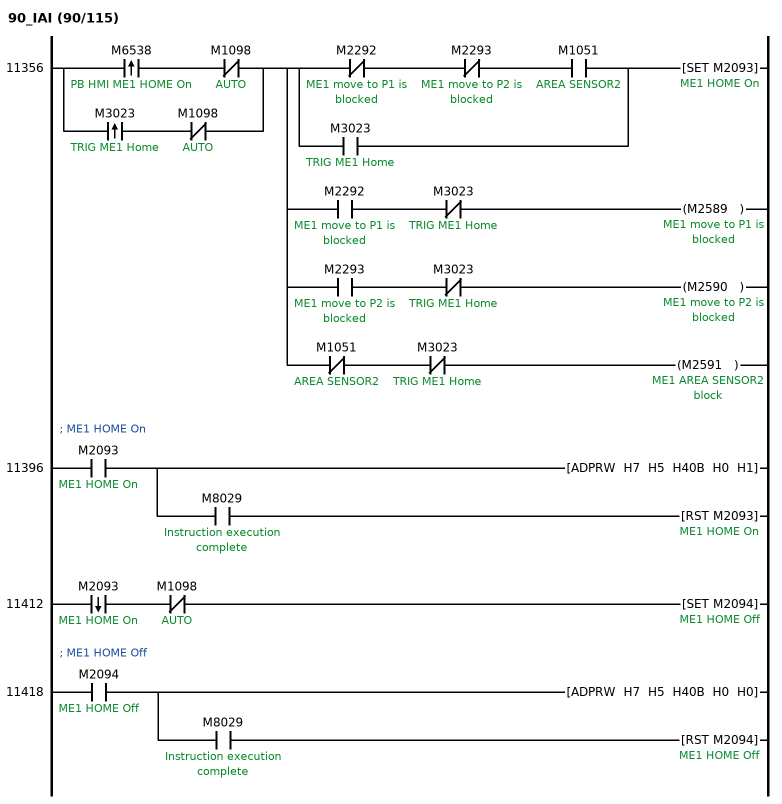
[picture p192: ladder of 90_IAI, rungs at steps 11356 to 11418]
11356 LDP     M6538  ; PB HMI ME1 HOME On
      ANI     M1098  ; AUTO
      LDP     M3023  ; TRIG ME1 Home
      ANI     M1098  ; AUTO
      ORB
      MPS
      LDI     M2292  ; ME1 move to P1 is blocked
      ANI     M2293  ; ME1 move to P2 is blocked
      AND     M1051  ; AREA SENSOR2
      OR      M3023  ; TRIG ME1 Home
      ANB
      SET     M2093  ; ME1 HOME On
      MRD
      AND     M2292  ; ME1 move to P1 is blocked
      ANI     M3023  ; TRIG ME1 Home
      OUT     M2589  ; ME1 move to P1 is blocked
      MRD
      AND     M2293  ; ME1 move to P2 is blocked
      ANI     M3023  ; TRIG ME1 Home
      OUT     M2590  ; ME1 move to P2 is blocked
      MPP
      ANI     M1051  ; AREA SENSOR2
      ANI     M3023  ; TRIG ME1 Home
      OUT     M2591  ; ME1 AREA SENSOR2 block
; ME1 HOME On
11396 LD      M2093  ; ME1 HOME On
      ADPRW   H7 H5 H40B H0 H1
      AND     M8029  ; Instruction execution complete
      RST     M2093  ; ME1 HOME On
11412 LDF     M2093  ; ME1 HOME On
      ANI     M1098  ; AUTO
      SET     M2094  ; ME1 HOME Off
; ME1 HOME Off
11418 LD      M2094  ; ME1 HOME Off
      ADPRW   H7 H5 H40B H0 H0
      AND     M8029  ; Instruction execution complete
      RST     M2094  ; ME1 HOME Off
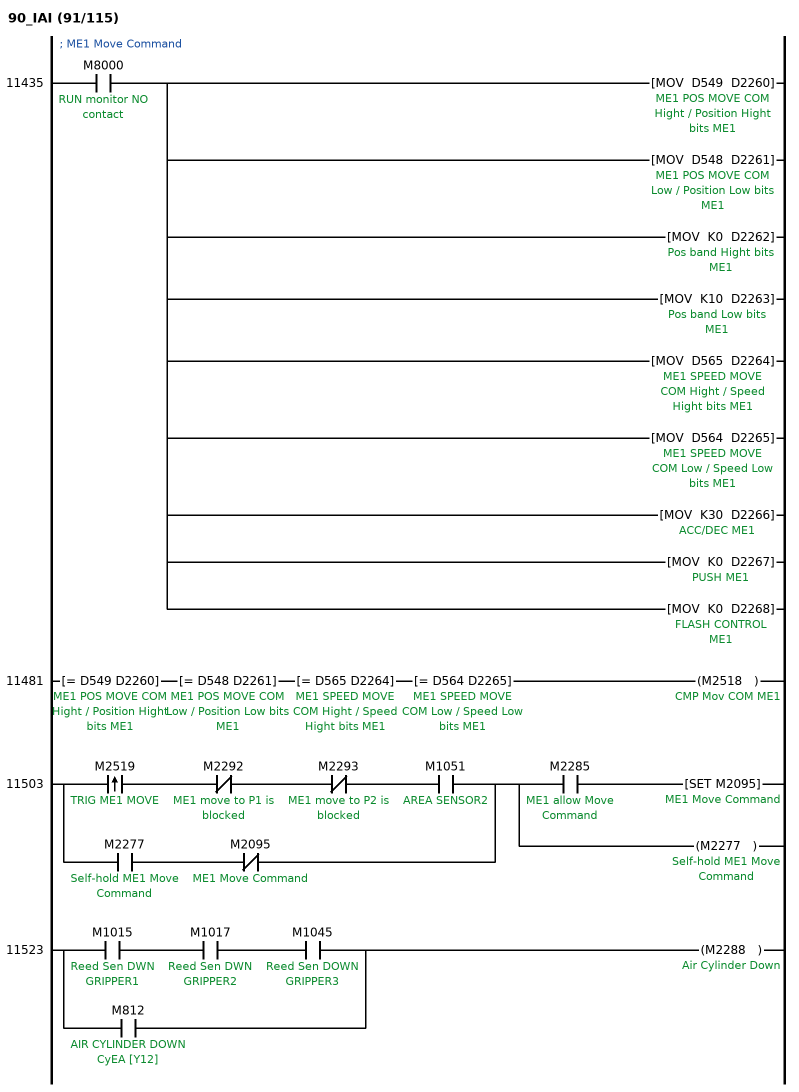
; ME1 Move Command
11435 LD      M8000  ; RUN monitor NO contact
      MOV     D549 D2260  ; ME1 POS MOVE COM Hight / Position Hight bits ME1
      MOV     D548 D2261  ; ME1 POS MOVE COM Low / Position Low bits ME1
      MOV     K0 D2262  ; Pos band Hight bits ME1
      MOV     K10 D2263  ; Pos band Low bits ME1
      MOV     D565 D2264  ; ME1 SPEED MOVE COM Hight / Speed Hight bits ME1
      MOV     D564 D2265  ; ME1 SPEED MOVE COM Low / Speed Low bits ME1
      MOV     K30 D2266  ; ACC/DEC ME1
      MOV     K0 D2267  ; PUSH ME1
      MOV     K0 D2268  ; FLASH CONTROL ME1
11481 LD=     D549 D2260  ; ME1 POS MOVE COM Hight / Position Hight bits ME1
      AND=    D548 D2261  ; ME1 POS MOVE COM Low / Position Low bits ME1
      AND=    D565 D2264  ; ME1 SPEED MOVE COM Hight / Speed Hight bits ME1
      AND=    D564 D2265  ; ME1 SPEED MOVE COM Low / Speed Low bits ME1
      OUT     M2518  ; CMP Mov COM ME1
11503 LDP     M2519  ; TRIG ME1 MOVE
      ANI     M2292  ; ME1 move to P1 is blocked
      ANI     M2293  ; ME1 move to P2 is blocked
      AND     M1051  ; AREA SENSOR2
      LD      M2277  ; Self-hold ME1 Move Command
      ANI     M2095  ; ME1 Move Command
      ORB
      MPS
      AND     M2285  ; ME1 allow Move Command
      SET     M2095  ; ME1 Move Command
      MPP
      OUT     M2277  ; Self-hold ME1 Move Command
11523 LD      M1015  ; Reed Sen DWN GRIPPER1
      AND     M1017  ; Reed Sen DWN GRIPPER2
      AND     M1045  ; Reed Sen DOWN GRIPPER3
      OR      M812  ; AIR CYLINDER DOWN CyEA [Y12]
      OUT     M2288  ; Air Cylinder Down
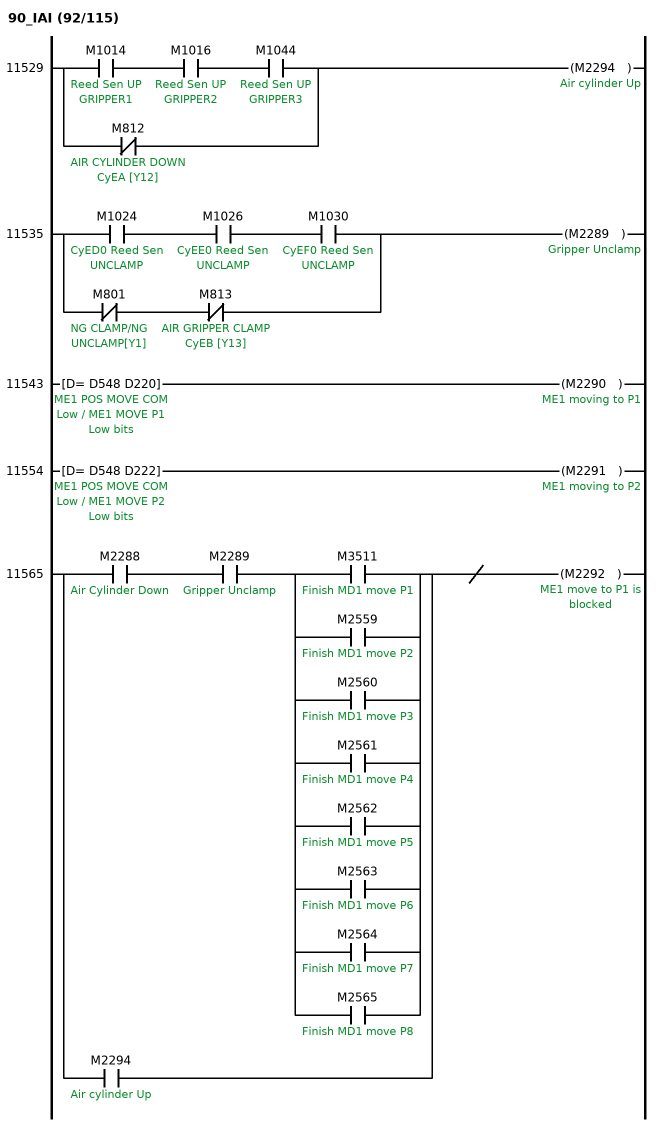
11529 LD      M1014  ; Reed Sen UP GRIPPER1
      AND     M1016  ; Reed Sen UP GRIPPER2
      AND     M1044  ; Reed Sen UP GRIPPER3
      ORI     M812  ; AIR CYLINDER DOWN CyEA [Y12]
      OUT     M2294  ; Air cylinder Up
11535 LD      M1024  ; CyED0 Reed Sen UNCLAMP
      AND     M1026  ; CyEE0 Reed Sen UNCLAMP
      AND     M1030  ; CyEF0 Reed Sen UNCLAMP
      LDI     M801  ; NG CLAMP/NG UNCLAMP[Y1]
      ANI     M813  ; AIR GRIPPER CLAMP CyEB [Y13]
      ORB
      OUT     M2289  ; Gripper Unclamp
11543 LDD=    D548 D220  ; ME1 POS MOVE COM Low / ME1 MOVE P1 Low bits
      OUT     M2290  ; ME1 moving to P1
11554 LDD=    D548 D222  ; ME1 POS MOVE COM Low / ME1 MOVE P2 Low bits
      OUT     M2291  ; ME1 moving to P2
11565 LD      M2288  ; Air Cylinder Down
      AND     M2289  ; Gripper Unclamp
      LD      M3511  ; Finish MD1 move P1
      OR      M2559  ; Finish MD1 move P2
      OR      M2560  ; Finish MD1 move P3
      OR      M2561  ; Finish MD1 move P4
      OR      M2562  ; Finish MD1 move P5
      OR      M2563  ; Finish MD1 move P6
      OR      M2564  ; Finish MD1 move P7
      OR      M2565  ; Finish MD1 move P8
      ANB
      OR      M2294  ; Air cylinder Up
      INV
      OUT     M2292  ; ME1 move to P1 is blocked
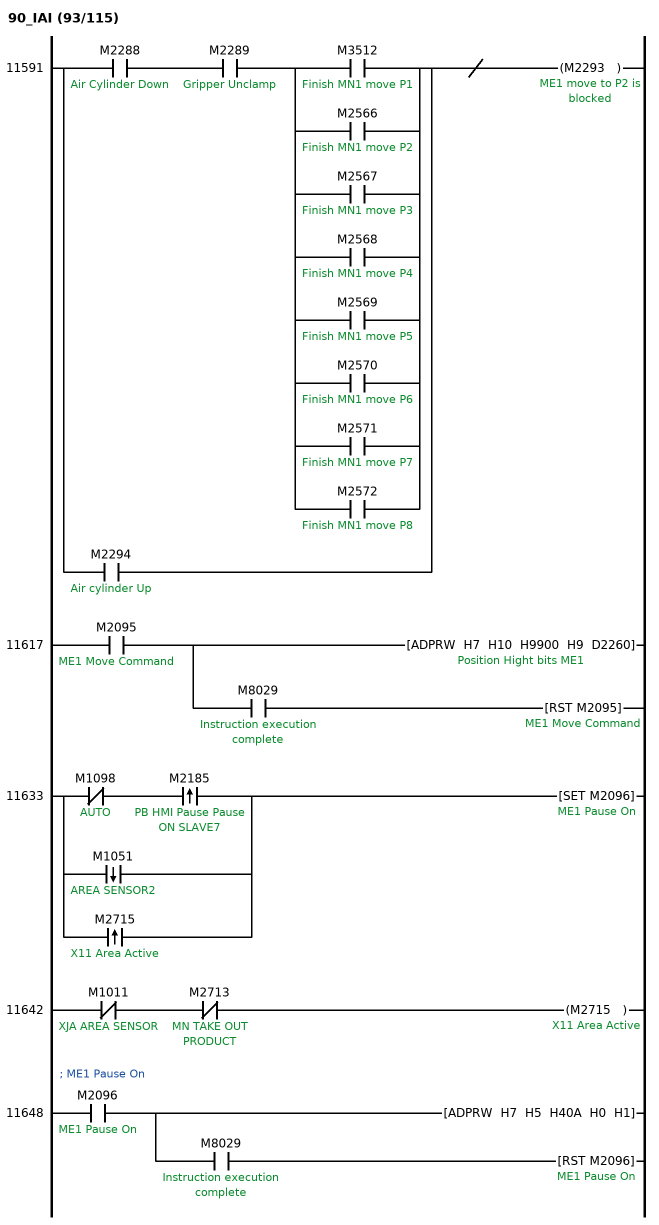
11591 LD      M2288  ; Air Cylinder Down
      AND     M2289  ; Gripper Unclamp
      LD      M3512  ; Finish MN1 move P1
      OR      M2566  ; Finish MN1 move P2
      OR      M2567  ; Finish MN1 move P3
      OR      M2568  ; Finish MN1 move P4
      OR      M2569  ; Finish MN1 move P5
      OR      M2570  ; Finish MN1 move P6
      OR      M2571  ; Finish MN1 move P7
      OR      M2572  ; Finish MN1 move P8
      ANB
      OR      M2294  ; Air cylinder Up
      INV
      OUT     M2293  ; ME1 move to P2 is blocked
11617 LD      M2095  ; ME1 Move Command
      ADPRW   H7 H10 H9900 H9 D2260
      AND     M8029  ; Instruction execution complete
      RST     M2095  ; ME1 Move Command
11633 LDI     M1098  ; AUTO
      ANDP    M2185  ; PB HMI Pause Pause ON SLAVE7
      ORF     M1051  ; AREA SENSOR2
      ORP     M2715  ; X11 Area Active
      SET     M2096  ; ME1 Pause On
11642 LDI     M1011  ; XJA AREA SENSOR
      ANI     M2713  ; MN TAKE OUT PRODUCT
      OUT     M2715  ; X11 Area Active
; ME1 Pause On
11648 LD      M2096  ; ME1 Pause On
      ADPRW   H7 H5 H40A H0 H1
      AND     M8029  ; Instruction execution complete
      RST     M2096  ; ME1 Pause On
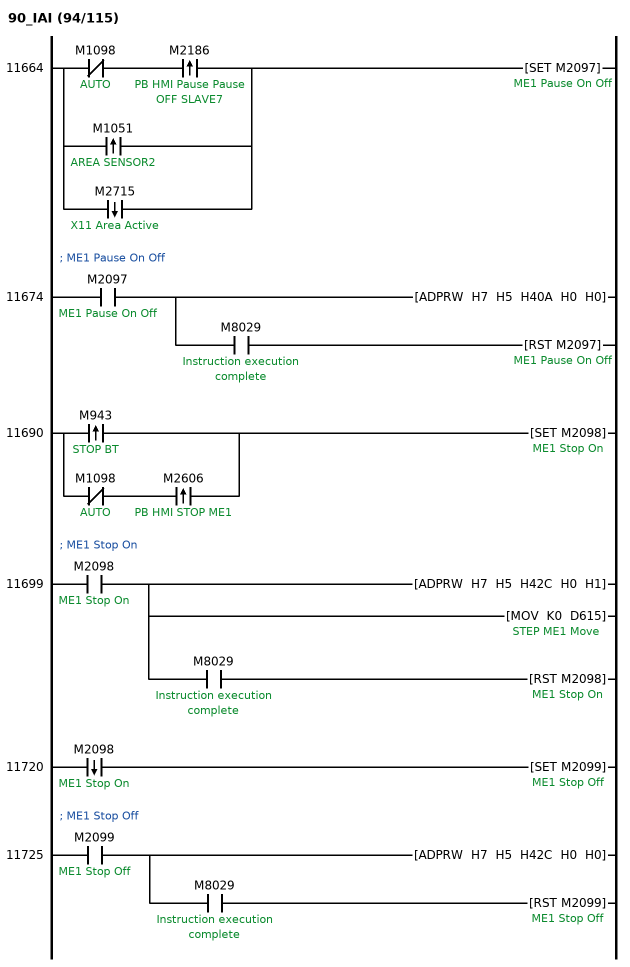
11664 LDI     M1098  ; AUTO
      ANDP    M2186  ; PB HMI Pause Pause OFF SLAVE7
      ORP     M1051  ; AREA SENSOR2
      ORF     M2715  ; X11 Area Active
      SET     M2097  ; ME1 Pause On Off
; ME1 Pause On Off
11674 LD      M2097  ; ME1 Pause On Off
      ADPRW   H7 H5 H40A H0 H0
      AND     M8029  ; Instruction execution complete
      RST     M2097  ; ME1 Pause On Off
11690 LDP     M943  ; STOP BT
      LDI     M1098  ; AUTO
      ANDP    M2606  ; PB HMI STOP ME1
      ORB
      SET     M2098  ; ME1 Stop On
; ME1 Stop On
11699 LD      M2098  ; ME1 Stop On
      ADPRW   H7 H5 H42C H0 H1
      MOV     K0 D615  ; STEP ME1 Move
      AND     M8029  ; Instruction execution complete
      RST     M2098  ; ME1 Stop On
11720 LDF     M2098  ; ME1 Stop On
      SET     M2099  ; ME1 Stop Off
; ME1 Stop Off
11725 LD      M2099  ; ME1 Stop Off
      ADPRW   H7 H5 H42C H0 H0
      AND     M8029  ; Instruction execution complete
      RST     M2099  ; ME1 Stop Off
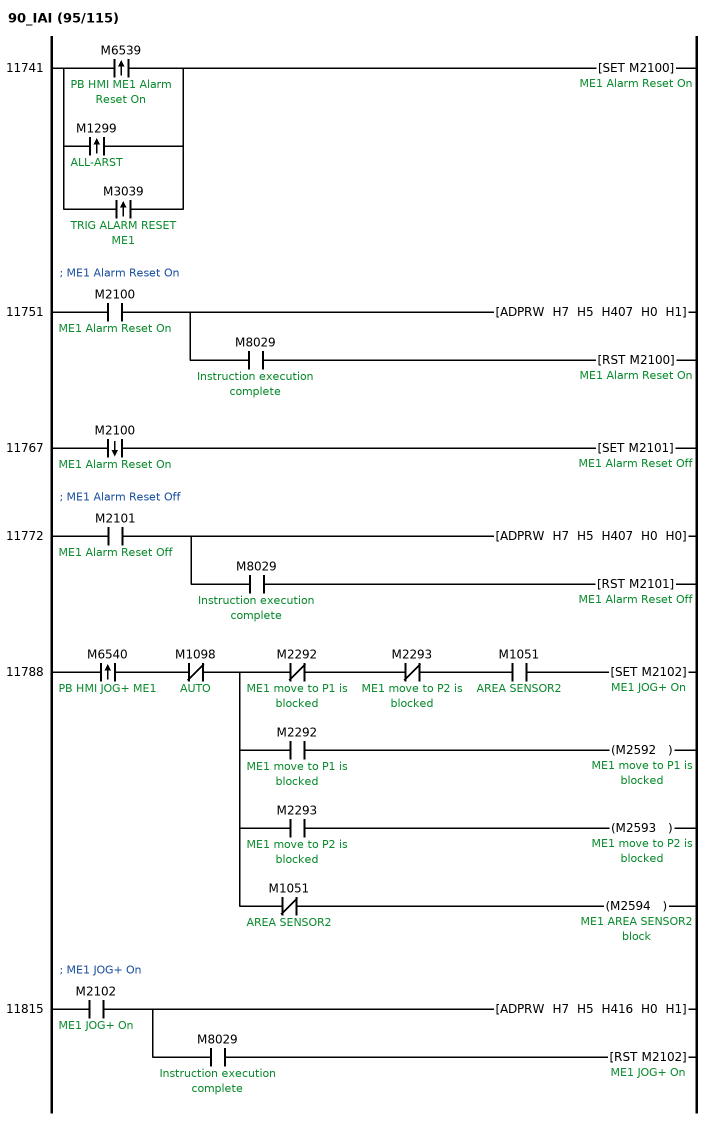
11741 LDP     M6539  ; PB HMI ME1 Alarm Reset On
      ORP     M1299  ; ALL-ARST
      ORP     M3039  ; TRIG ALARM RESET ME1
      SET     M2100  ; ME1 Alarm Reset On
; ME1 Alarm Reset On
11751 LD      M2100  ; ME1 Alarm Reset On
      ADPRW   H7 H5 H407 H0 H1
      AND     M8029  ; Instruction execution complete
      RST     M2100  ; ME1 Alarm Reset On
11767 LDF     M2100  ; ME1 Alarm Reset On
      SET     M2101  ; ME1 Alarm Reset Off
; ME1 Alarm Reset Off
11772 LD      M2101  ; ME1 Alarm Reset Off
      ADPRW   H7 H5 H407 H0 H0
      AND     M8029  ; Instruction execution complete
      RST     M2101  ; ME1 Alarm Reset Off
11788 LDP     M6540  ; PB HMI JOG+ ME1
      ANI     M1098  ; AUTO
      MPS
      ANI     M2292  ; ME1 move to P1 is blocked
      ANI     M2293  ; ME1 move to P2 is blocked
      AND     M1051  ; AREA SENSOR2
      SET     M2102  ; ME1 JOG+ On
      MRD
      AND     M2292  ; ME1 move to P1 is blocked
      OUT     M2592  ; ME1 move to P1 is blocked
      MRD
      AND     M2293  ; ME1 move to P2 is blocked
      OUT     M2593  ; ME1 move to P2 is blocked
      MPP
      ANI     M1051  ; AREA SENSOR2
      OUT     M2594  ; ME1 AREA SENSOR2 block
; ME1 JOG+ On
11815 LD      M2102  ; ME1 JOG+ On
      ADPRW   H7 H5 H416 H0 H1
      AND     M8029  ; Instruction execution complete
      RST     M2102  ; ME1 JOG+ On
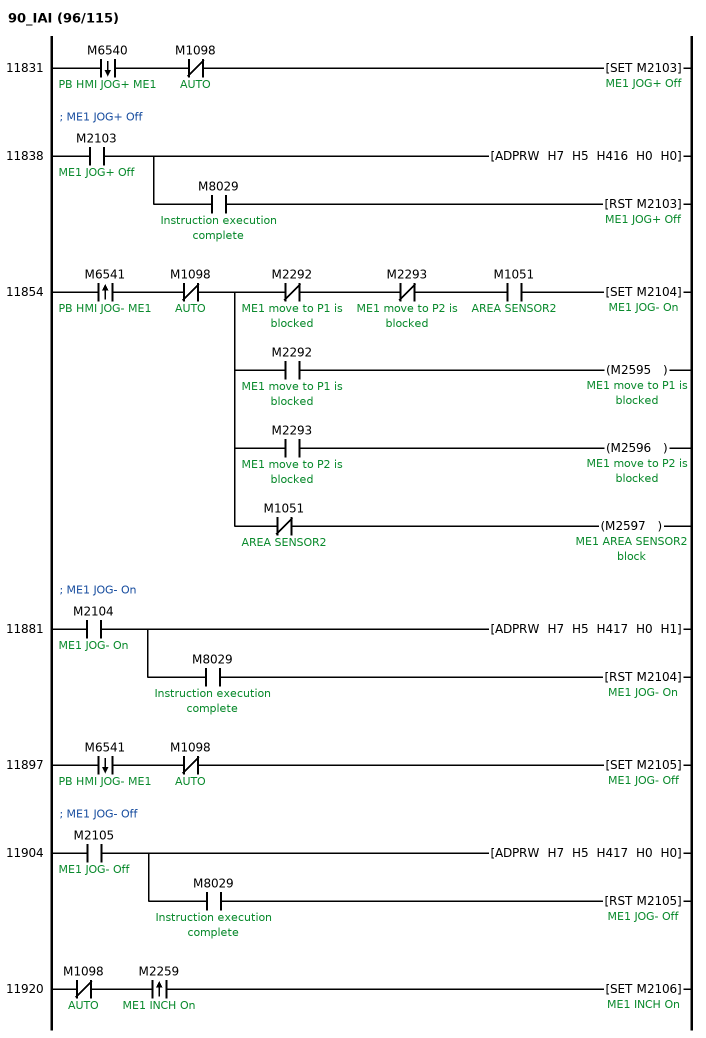
11831 LDF     M6540  ; PB HMI JOG+ ME1
      ANI     M1098  ; AUTO
      SET     M2103  ; ME1 JOG+ Off
; ME1 JOG+ Off
11838 LD      M2103  ; ME1 JOG+ Off
      ADPRW   H7 H5 H416 H0 H0
      AND     M8029  ; Instruction execution complete
      RST     M2103  ; ME1 JOG+ Off
11854 LDP     M6541  ; PB HMI JOG- ME1
      ANI     M1098  ; AUTO
      MPS
      ANI     M2292  ; ME1 move to P1 is blocked
      ANI     M2293  ; ME1 move to P2 is blocked
      AND     M1051  ; AREA SENSOR2
      SET     M2104  ; ME1 JOG- On
      MRD
      AND     M2292  ; ME1 move to P1 is blocked
      OUT     M2595  ; ME1 move to P1 is blocked
      MRD
      AND     M2293  ; ME1 move to P2 is blocked
      OUT     M2596  ; ME1 move to P2 is blocked
      MPP
      ANI     M1051  ; AREA SENSOR2
      OUT     M2597  ; ME1 AREA SENSOR2 block
; ME1 JOG- On
11881 LD      M2104  ; ME1 JOG- On
      ADPRW   H7 H5 H417 H0 H1
      AND     M8029  ; Instruction execution complete
      RST     M2104  ; ME1 JOG- On
11897 LDF     M6541  ; PB HMI JOG- ME1
      ANI     M1098  ; AUTO
      SET     M2105  ; ME1 JOG- Off
; ME1 JOG- Off
11904 LD      M2105  ; ME1 JOG- Off
      ADPRW   H7 H5 H417 H0 H0
      AND     M8029  ; Instruction execution complete
      RST     M2105  ; ME1 JOG- Off
11920 LDI     M1098  ; AUTO
      ANDP    M2259  ; ME1 INCH On
      SET     M2106  ; ME1 INCH On
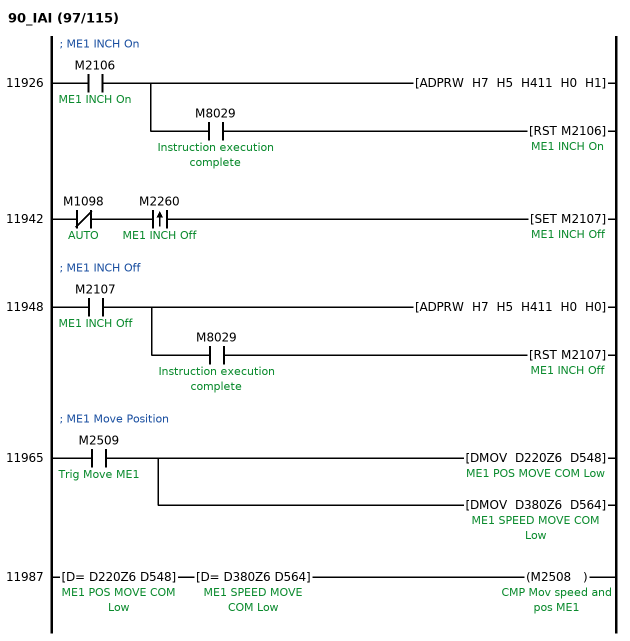
; ME1 INCH On
11926 LD      M2106  ; ME1 INCH On
      ADPRW   H7 H5 H411 H0 H1
      AND     M8029  ; Instruction execution complete
      RST     M2106  ; ME1 INCH On
11942 LDI     M1098  ; AUTO
      ANDP    M2260  ; ME1 INCH Off
      SET     M2107  ; ME1 INCH Off
; ME1 INCH Off
11948 LD      M2107  ; ME1 INCH Off
      ADPRW   H7 H5 H411 H0 H0
      AND     M8029  ; Instruction execution complete
      RST     M2107  ; ME1 INCH Off
; ME1 Move Position
11965 LD      M2509  ; Trig Move ME1
      DMOV    D220Z6 D548
        [note] Position
      DMOV    D380Z6 D564
        [note] Speed
11987 LDD=    D220Z6 D548  ; ME1 POS MOVE COM Low
      ANDD=   D380Z6 D564  ; ME1 SPEED MOVE COM Low
      OUT     M2508  ; CMP Mov speed and pos ME1
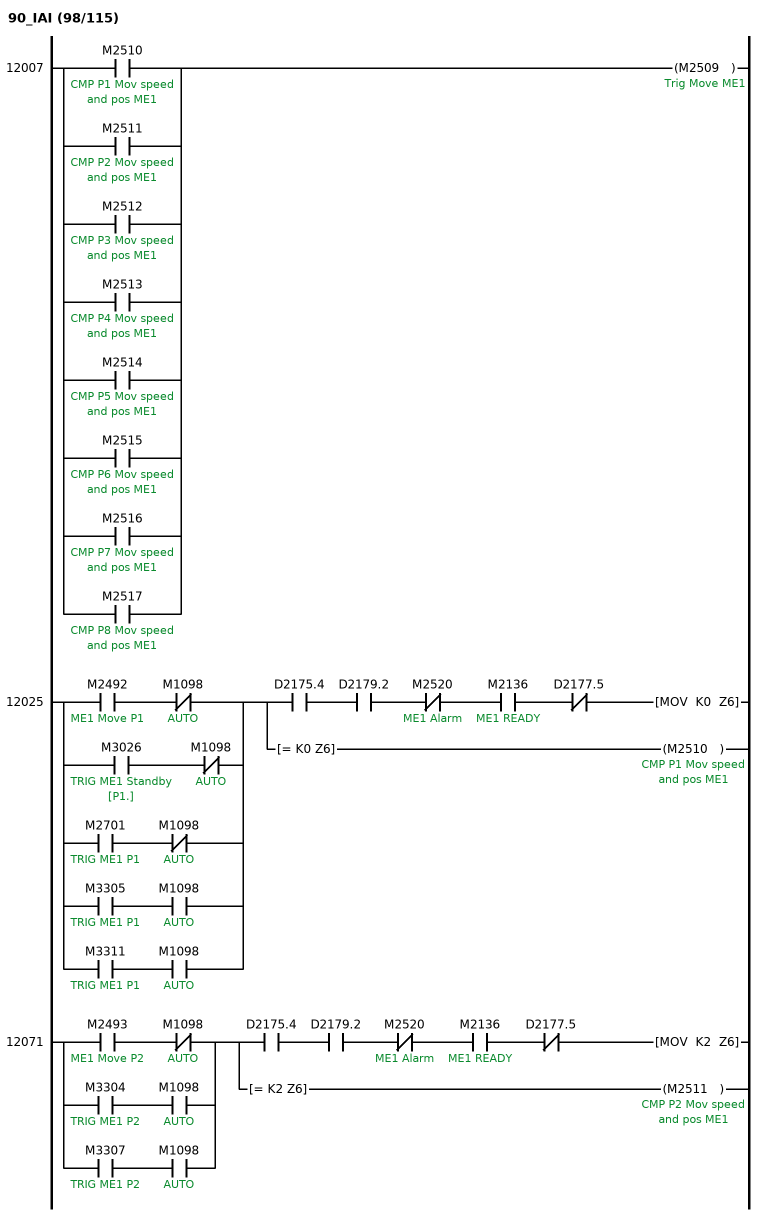
12007 LD      M2510  ; CMP P1 Mov speed and pos ME1
      OR      M2511  ; CMP P2 Mov speed and pos ME1
      OR      M2512  ; CMP P3 Mov speed and pos ME1
      OR      M2513  ; CMP P4 Mov speed and pos ME1
      OR      M2514  ; CMP P5 Mov speed and pos ME1
      OR      M2515  ; CMP P6 Mov speed and pos ME1
      OR      M2516  ; CMP P7 Mov speed and pos ME1
      OR      M2517  ; CMP P8 Mov speed and pos ME1
      OUT     M2509  ; Trig Move ME1
12025 LD      M2492  ; ME1 Move P1
      ANI     M1098  ; AUTO
      LD      M3026  ; TRIG ME1 Standby [P1.]
      ANI     M1098  ; AUTO
      ORB
      LD      M2701  ; TRIG ME1 P1
      ANI     M1098  ; AUTO
      ORB
      LD      M3305  ; TRIG ME1 P1
      AND     M1098  ; AUTO
      ORB
      LD      M3311  ; TRIG ME1 P1
      AND     M1098  ; AUTO
      ORB
      MPS
      AND     D2175.4
      AND     D2179.2
      ANI     M2520  ; ME1 Alarm
      AND     M2136  ; ME1 READY
      ANI     D2177.5
      MOV     K0 Z6
      MPP
      AND=    K0 Z6
      OUT     M2510  ; CMP P1 Mov speed and pos ME1
12071 LD      M2493  ; ME1 Move P2
      ANI     M1098  ; AUTO
      LD      M3304  ; TRIG ME1 P2
      AND     M1098  ; AUTO
      ORB
      LD      M3307  ; TRIG ME1 P2
      AND     M1098  ; AUTO
      ORB
      MPS
      AND     D2175.4
      AND     D2179.2
      ANI     M2520  ; ME1 Alarm
      AND     M2136  ; ME1 READY
      ANI     D2177.5
      MOV     K2 Z6
      MPP
      AND=    K2 Z6
      OUT     M2511  ; CMP P2 Mov speed and pos ME1
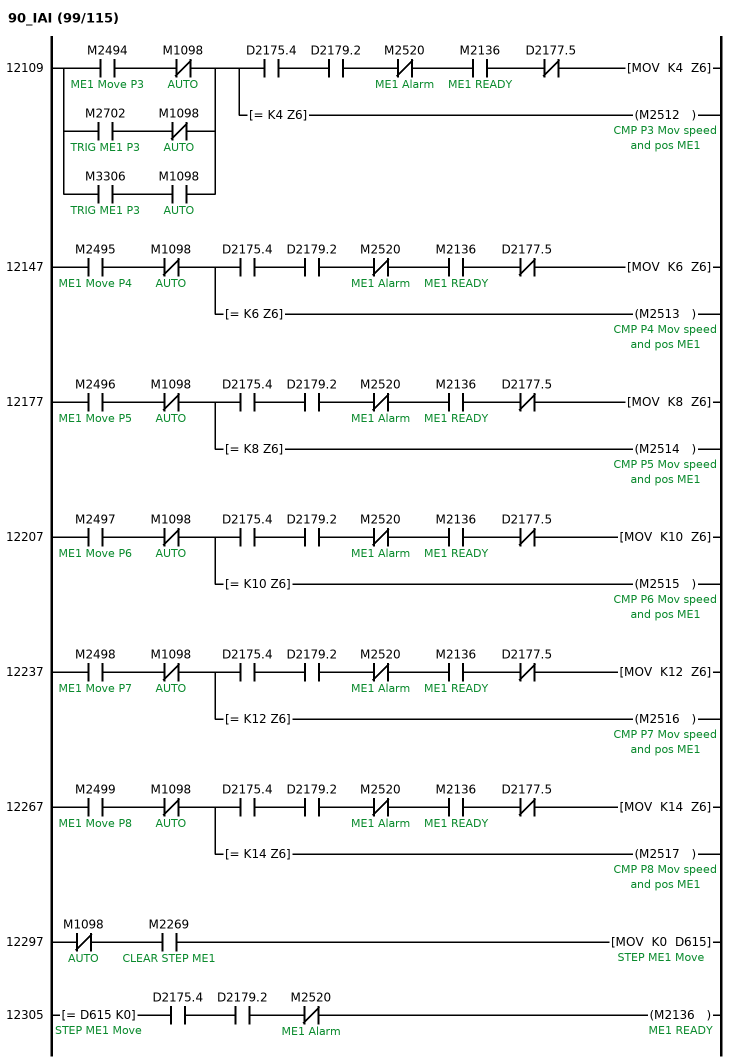
12109 LD      M2494  ; ME1 Move P3
      ANI     M1098  ; AUTO
      LD      M2702  ; TRIG ME1 P3
      ANI     M1098  ; AUTO
      ORB
      LD      M3306  ; TRIG ME1 P3
      AND     M1098  ; AUTO
      ORB
      MPS
      AND     D2175.4
      AND     D2179.2
      ANI     M2520  ; ME1 Alarm
      AND     M2136  ; ME1 READY
      ANI     D2177.5
      MOV     K4 Z6
      MPP
      AND=    K4 Z6
      OUT     M2512  ; CMP P3 Mov speed and pos ME1
12147 LD      M2495  ; ME1 Move P4
      ANI     M1098  ; AUTO
      MPS
      AND     D2175.4
      AND     D2179.2
      ANI     M2520  ; ME1 Alarm
      AND     M2136  ; ME1 READY
      ANI     D2177.5
      MOV     K6 Z6
      MPP
      AND=    K6 Z6
      OUT     M2513  ; CMP P4 Mov speed and pos ME1
12177 LD      M2496  ; ME1 Move P5
      ANI     M1098  ; AUTO
      MPS
      AND     D2175.4
      AND     D2179.2
      ANI     M2520  ; ME1 Alarm
      AND     M2136  ; ME1 READY
      ANI     D2177.5
      MOV     K8 Z6
      MPP
      AND=    K8 Z6
      OUT     M2514  ; CMP P5 Mov speed and pos ME1
12207 LD      M2497  ; ME1 Move P6
      ANI     M1098  ; AUTO
      MPS
      AND     D2175.4
      AND     D2179.2
      ANI     M2520  ; ME1 Alarm
      AND     M2136  ; ME1 READY
      ANI     D2177.5
      MOV     K10 Z6
      MPP
      AND=    K10 Z6
      OUT     M2515  ; CMP P6 Mov speed and pos ME1
12237 LD      M2498  ; ME1 Move P7
      ANI     M1098  ; AUTO
      MPS
      AND     D2175.4
      AND     D2179.2
      ANI     M2520  ; ME1 Alarm
      AND     M2136  ; ME1 READY
      ANI     D2177.5
      MOV     K12 Z6
      MPP
      AND=    K12 Z6
      OUT     M2516  ; CMP P7 Mov speed and pos ME1
12267 LD      M2499  ; ME1 Move P8
      ANI     M1098  ; AUTO
      MPS
      AND     D2175.4
      AND     D2179.2
      ANI     M2520  ; ME1 Alarm
      AND     M2136  ; ME1 READY
      ANI     D2177.5
      MOV     K14 Z6
      MPP
      AND=    K14 Z6
      OUT     M2517  ; CMP P8 Mov speed and pos ME1
12297 LDI     M1098  ; AUTO
      AND     M2269  ; CLEAR STEP ME1
      MOV     K0 D615
12305 LD=     D615 K0  ; STEP ME1 Move
      AND     D2175.4
      AND     D2179.2
      ANI     M2520  ; ME1 Alarm
      OUT     M2136  ; ME1 READY
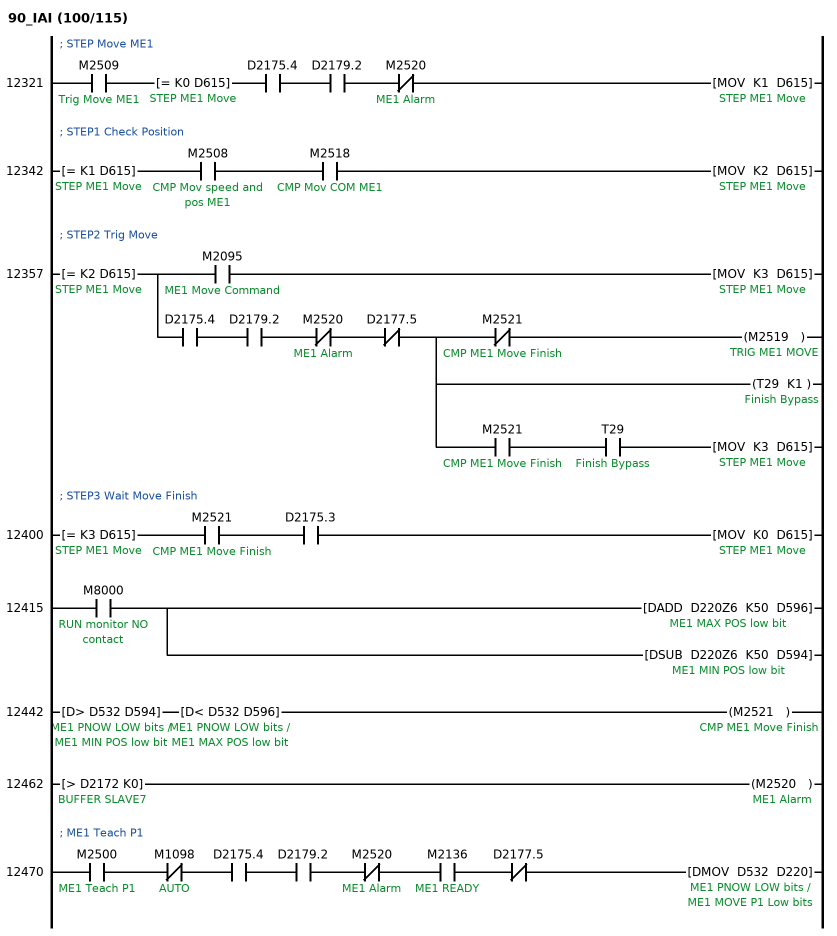
; STEP Move ME1
12321 LD      M2509  ; Trig Move ME1
      AND=    K0 D615  ; STEP ME1 Move
      AND     D2175.4
      AND     D2179.2
      ANI     M2520  ; ME1 Alarm
      MOV     K1 D615
; STEP1 Check Position
12342 LD=     K1 D615  ; STEP ME1 Move
      AND     M2508  ; CMP Mov speed and pos ME1
      AND     M2518  ; CMP Mov COM ME1
      MOV     K2 D615
; STEP2 Trig Move
12357 LD=     K2 D615  ; STEP ME1 Move
      MPS
      AND     M2095  ; ME1 Move Command
      MOV     K3 D615
      MPP
      AND     D2175.4
      AND     D2179.2
      ANI     M2520  ; ME1 Alarm
      ANI     D2177.5
      MPS
      ANI     M2521  ; CMP ME1 Move Finish
      OUT     M2519  ; TRIG ME1 MOVE
      MPP
      OUT     T29 K1  ; Finish Bypass
      AND     M2521  ; CMP ME1 Move Finish
      AND     T29  ; Finish Bypass
      MOV     K3 D615
; STEP3 Wait Move Finish
12400 LD=     K3 D615  ; STEP ME1 Move
      AND     M2521  ; CMP ME1 Move Finish
      AND     D2175.3
      MOV     K0 D615
12415 LD      M8000  ; RUN monitor NO contact
      DADD    D220Z6 K50 D596  ; ME1 MAX POS low bit
      DSUB    D220Z6 K50 D594  ; ME1 MIN POS low bit
12442 LDD>    D532 D594  ; ME1 PNOW LOW bits / ME1 MIN POS low bit
      ANDD<   D532 D596  ; ME1 PNOW LOW bits / ME1 MAX POS low bit
      OUT     M2521  ; CMP ME1 Move Finish
12462 LD>     D2172 K0  ; BUFFER SLAVE7
      OUT     M2520  ; ME1 Alarm
; ME1 Teach P1
12470 LD      M2500  ; ME1 Teach P1
      ANI     M1098  ; AUTO
      AND     D2175.4
      AND     D2179.2
      ANI     M2520  ; ME1 Alarm
      AND     M2136  ; ME1 READY
      ANI     D2177.5
      DMOV    D532 D220
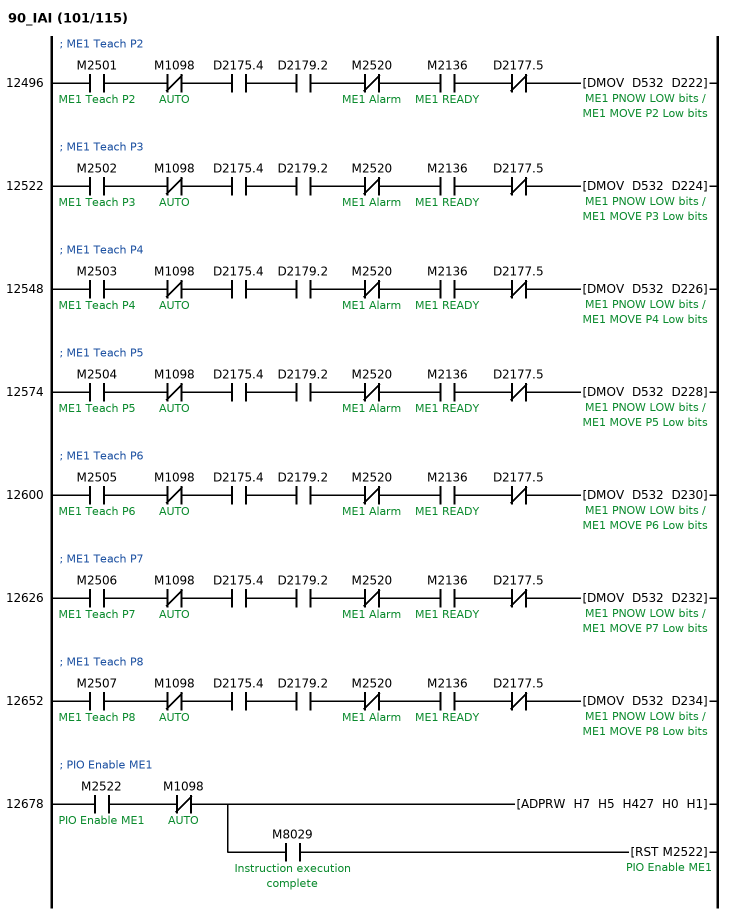
; ME1 Teach P2
12496 LD      M2501  ; ME1 Teach P2
      ANI     M1098  ; AUTO
      AND     D2175.4
      AND     D2179.2
      ANI     M2520  ; ME1 Alarm
      AND     M2136  ; ME1 READY
      ANI     D2177.5
      DMOV    D532 D222
; ME1 Teach P3
12522 LD      M2502  ; ME1 Teach P3
      ANI     M1098  ; AUTO
      AND     D2175.4
      AND     D2179.2
      ANI     M2520  ; ME1 Alarm
      AND     M2136  ; ME1 READY
      ANI     D2177.5
      DMOV    D532 D224  ; ME1 MOVE P3 Low bits
; ME1 Teach P4
12548 LD      M2503  ; ME1 Teach P4
      ANI     M1098  ; AUTO
      AND     D2175.4
      AND     D2179.2
      ANI     M2520  ; ME1 Alarm
      AND     M2136  ; ME1 READY
      ANI     D2177.5
      DMOV    D532 D226  ; ME1 MOVE P4 Low bits
; ME1 Teach P5
12574 LD      M2504  ; ME1 Teach P5
      ANI     M1098  ; AUTO
      AND     D2175.4
      AND     D2179.2
      ANI     M2520  ; ME1 Alarm
      AND     M2136  ; ME1 READY
      ANI     D2177.5
      DMOV    D532 D228  ; ME1 MOVE P5 Low bits
; ME1 Teach P6
12600 LD      M2505  ; ME1 Teach P6
      ANI     M1098  ; AUTO
      AND     D2175.4
      AND     D2179.2
      ANI     M2520  ; ME1 Alarm
      AND     M2136  ; ME1 READY
      ANI     D2177.5
      DMOV    D532 D230  ; ME1 MOVE P6 Low bits
; ME1 Teach P7
12626 LD      M2506  ; ME1 Teach P7
      ANI     M1098  ; AUTO
      AND     D2175.4
      AND     D2179.2
      ANI     M2520  ; ME1 Alarm
      AND     M2136  ; ME1 READY
      ANI     D2177.5
      DMOV    D532 D232  ; ME1 MOVE P7 Low bits
; ME1 Teach P8
12652 LD      M2507  ; ME1 Teach P8
      ANI     M1098  ; AUTO
      AND     D2175.4
      AND     D2179.2
      ANI     M2520  ; ME1 Alarm
      AND     M2136  ; ME1 READY
      ANI     D2177.5
      DMOV    D532 D234  ; ME1 MOVE P8 Low bits
; PIO Enable ME1
12678 LD      M2522  ; PIO Enable ME1
      ANI     M1098  ; AUTO
      ADPRW   H7 H5 H427 H0 H1
      AND     M8029  ; Instruction execution complete
      RST     M2522  ; PIO Enable ME1
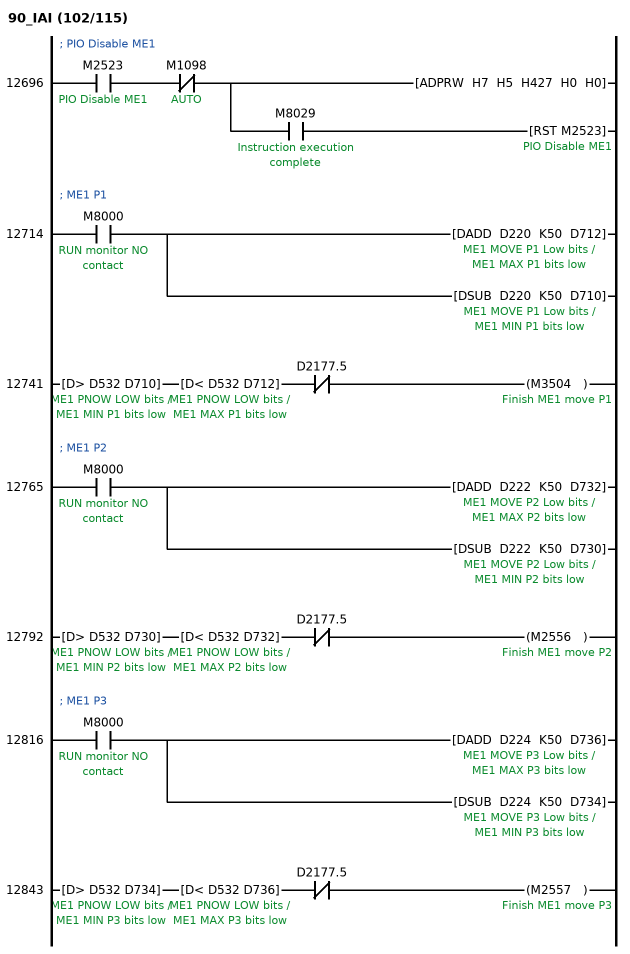
; PIO Disable ME1
12696 LD      M2523  ; PIO Disable ME1
      ANI     M1098  ; AUTO
      ADPRW   H7 H5 H427 H0 H0
      AND     M8029  ; Instruction execution complete
      RST     M2523  ; PIO Disable ME1
; ME1 P1
12714 LD      M8000  ; RUN monitor NO contact
      DADD    D220 K50 D712  ; ME1 MAX P1 bits low
      DSUB    D220 K50 D710  ; ME1 MIN P1 bits low
12741 LDD>    D532 D710  ; ME1 PNOW LOW bits / ME1 MIN P1 bits low
      ANDD<   D532 D712  ; ME1 PNOW LOW bits / ME1 MAX P1 bits low
      ANI     D2177.5
      OUT     M3504  ; Finish ME1 move P1
; ME1 P2
12765 LD      M8000  ; RUN monitor NO contact
      DADD    D222 K50 D732  ; ME1 MAX P2 bits low
      DSUB    D222 K50 D730  ; ME1 MIN P2 bits low
12792 LDD>    D532 D730  ; ME1 PNOW LOW bits / ME1 MIN P2 bits low
      ANDD<   D532 D732  ; ME1 PNOW LOW bits / ME1 MAX P2 bits low
      ANI     D2177.5
      OUT     M2556  ; Finish ME1 move P2
; ME1 P3
12816 LD      M8000  ; RUN monitor NO contact
      DADD    D224 K50 D736  ; ME1 MAX P3 bits low
      DSUB    D224 K50 D734  ; ME1 MIN P3 bits low
12843 LDD>    D532 D734  ; ME1 PNOW LOW bits / ME1 MIN P3 bits low
      ANDD<   D532 D736  ; ME1 PNOW LOW bits / ME1 MAX P3 bits low
      ANI     D2177.5
      OUT     M2557  ; Finish ME1 move P3
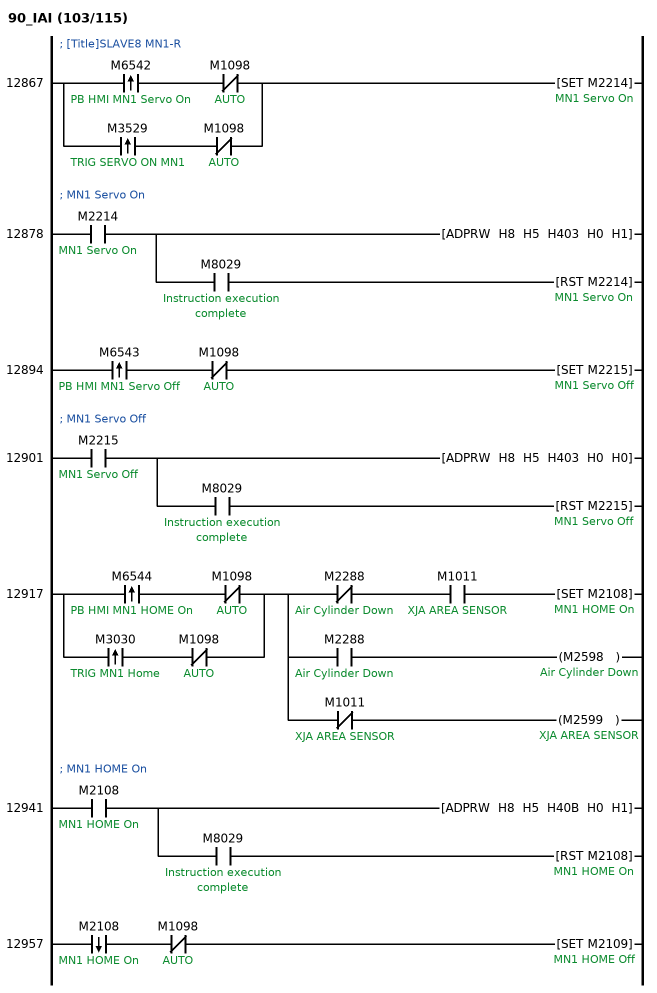
; [Title]SLAVE8 MN1-R
12867 LDP     M6542  ; PB HMI MN1 Servo On
      ANI     M1098  ; AUTO
      LDP     M3529  ; TRIG SERVO ON MN1
      ANI     M1098  ; AUTO
      ORB
      SET     M2214  ; MN1 Servo On
; MN1 Servo On
12878 LD      M2214  ; MN1 Servo On
      ADPRW   H8 H5 H403 H0 H1
      AND     M8029  ; Instruction execution complete
      RST     M2214  ; MN1 Servo On
12894 LDP     M6543  ; PB HMI MN1 Servo Off
      ANI     M1098  ; AUTO
      SET     M2215  ; MN1 Servo Off
; MN1 Servo Off
12901 LD      M2215  ; MN1 Servo Off
      ADPRW   H8 H5 H403 H0 H0
      AND     M8029  ; Instruction execution complete
      RST     M2215  ; MN1 Servo Off
12917 LDP     M6544  ; PB HMI MN1 HOME On
      ANI     M1098  ; AUTO
      LDP     M3030  ; TRIG MN1 Home
      ANI     M1098  ; AUTO
      ORB
      MPS
      ANI     M2288  ; Air Cylinder Down
      AND     M1011  ; XJA AREA SENSOR
      SET     M2108  ; MN1 HOME On
      MRD
      AND     M2288  ; Air Cylinder Down
      OUT     M2598  ; Air Cylinder Down
      MPP
      ANI     M1011  ; XJA AREA SENSOR
      OUT     M2599  ; XJA AREA SENSOR
; MN1 HOME On
12941 LD      M2108  ; MN1 HOME On
      ADPRW   H8 H5 H40B H0 H1
      AND     M8029  ; Instruction execution complete
      RST     M2108  ; MN1 HOME On
12957 LDF     M2108  ; MN1 HOME On
      ANI     M1098  ; AUTO
      SET     M2109  ; MN1 HOME Off
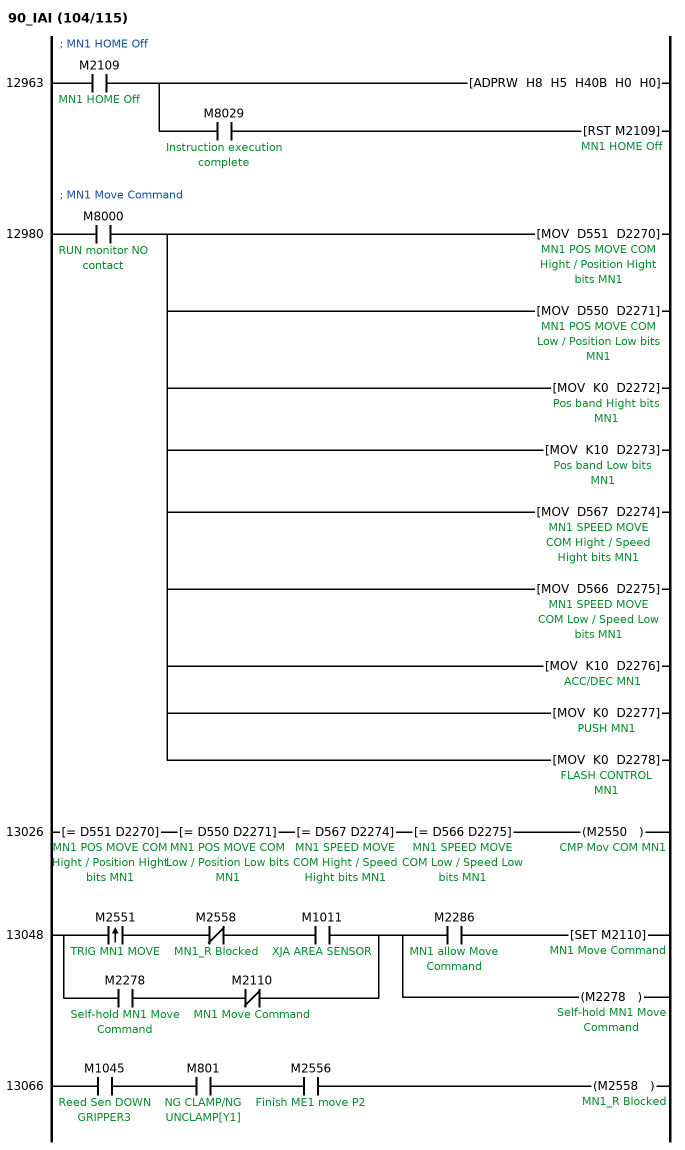
; MN1 HOME Off
12963 LD      M2109  ; MN1 HOME Off
      ADPRW   H8 H5 H40B H0 H0
      AND     M8029  ; Instruction execution complete
      RST     M2109  ; MN1 HOME Off
; MN1 Move Command
12980 LD      M8000  ; RUN monitor NO contact
      MOV     D551 D2270  ; MN1 POS MOVE COM Hight / Position Hight bits MN1
      MOV     D550 D2271  ; MN1 POS MOVE COM Low / Position Low bits MN1
      MOV     K0 D2272  ; Pos band Hight bits MN1
      MOV     K10 D2273  ; Pos band Low bits MN1
      MOV     D567 D2274  ; MN1 SPEED MOVE COM Hight / Speed Hight bits MN1
      MOV     D566 D2275  ; MN1 SPEED MOVE COM Low / Speed Low bits MN1
      MOV     K10 D2276  ; ACC/DEC MN1
      MOV     K0 D2277  ; PUSH MN1
      MOV     K0 D2278  ; FLASH CONTROL MN1
13026 LD=     D551 D2270  ; MN1 POS MOVE COM Hight / Position Hight bits MN1
      AND=    D550 D2271  ; MN1 POS MOVE COM Low / Position Low bits MN1
      AND=    D567 D2274  ; MN1 SPEED MOVE COM Hight / Speed Hight bits MN1
      AND=    D566 D2275  ; MN1 SPEED MOVE COM Low / Speed Low bits MN1
      OUT     M2550  ; CMP Mov COM MN1
13048 LDP     M2551  ; TRIG MN1 MOVE
      ANI     M2558  ; MN1_R Blocked
      AND     M1011  ; XJA AREA SENSOR
      LD      M2278  ; Self-hold MN1 Move Command
      ANI     M2110  ; MN1 Move Command
      ORB
      MPS
      AND     M2286  ; MN1 allow Move Command
      SET     M2110  ; MN1 Move Command
      MPP
      OUT     M2278  ; Self-hold MN1 Move Command
13066 LD      M1045  ; Reed Sen DOWN GRIPPER3
      AND     M801  ; NG CLAMP/NG UNCLAMP[Y1]
      AND     M2556  ; Finish ME1 move P2
      OUT     M2558  ; MN1_R Blocked
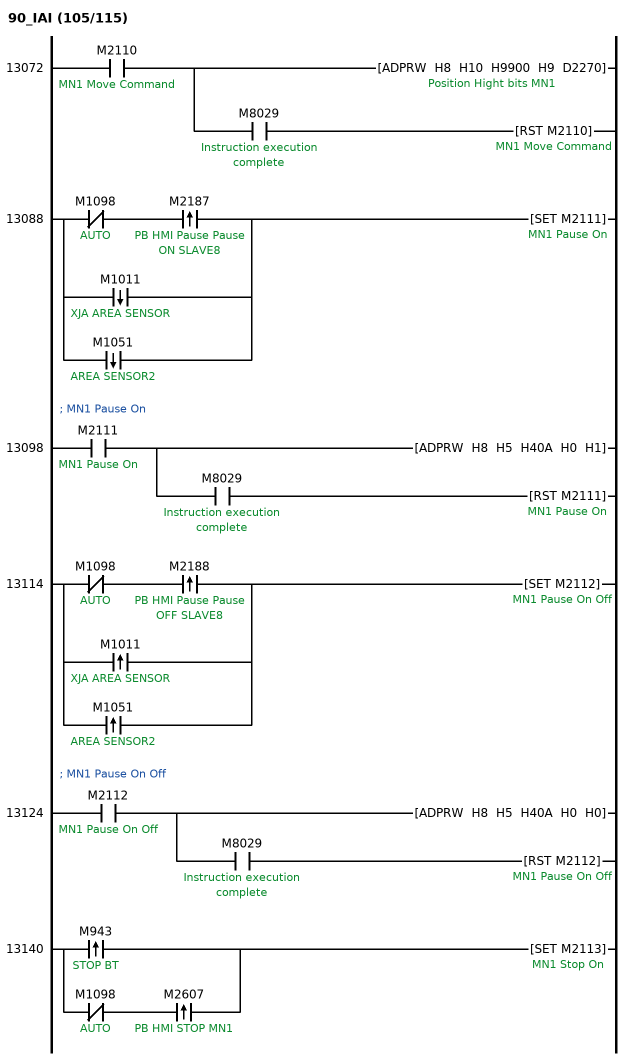
13072 LD      M2110  ; MN1 Move Command
      ADPRW   H8 H10 H9900 H9 D2270
      AND     M8029  ; Instruction execution complete
      RST     M2110  ; MN1 Move Command
13088 LDI     M1098  ; AUTO
      ANDP    M2187  ; PB HMI Pause Pause ON SLAVE8
      ORF     M1011  ; XJA AREA SENSOR
      ORF     M1051  ; AREA SENSOR2
      SET     M2111  ; MN1 Pause On
; MN1 Pause On
13098 LD      M2111  ; MN1 Pause On
      ADPRW   H8 H5 H40A H0 H1
      AND     M8029  ; Instruction execution complete
      RST     M2111  ; MN1 Pause On
13114 LDI     M1098  ; AUTO
      ANDP    M2188  ; PB HMI Pause Pause OFF SLAVE8
      ORP     M1011  ; XJA AREA SENSOR
      ORP     M1051  ; AREA SENSOR2
      SET     M2112  ; MN1 Pause On Off
; MN1 Pause On Off
13124 LD      M2112  ; MN1 Pause On Off
      ADPRW   H8 H5 H40A H0 H0
      AND     M8029  ; Instruction execution complete
      RST     M2112  ; MN1 Pause On Off
13140 LDP     M943  ; STOP BT
      LDI     M1098  ; AUTO
      ANDP    M2607  ; PB HMI STOP MN1
      ORB
      SET     M2113  ; MN1 Stop On
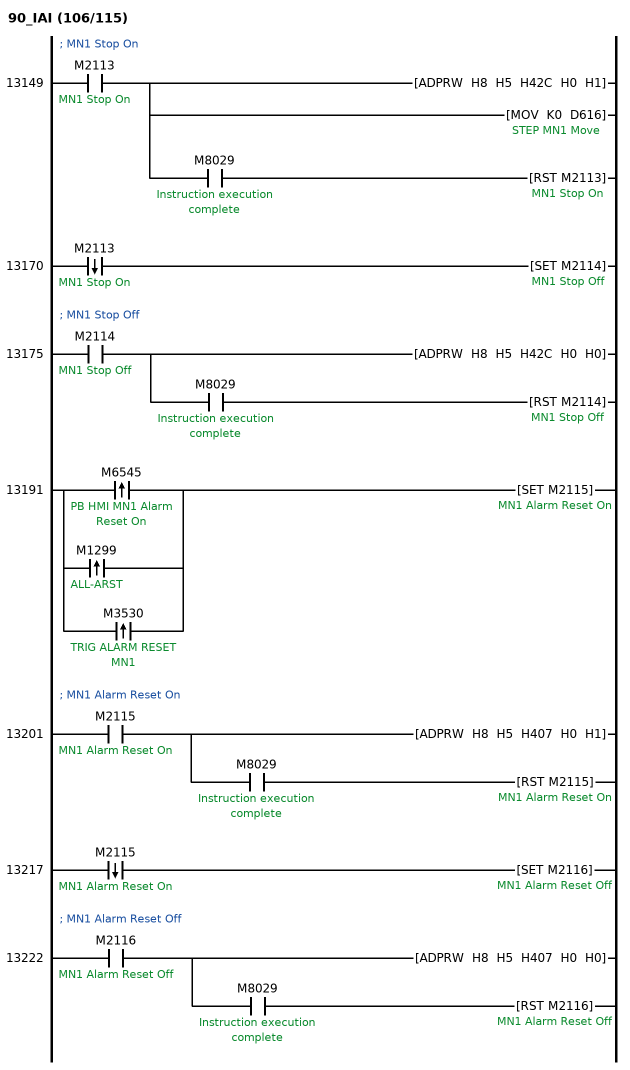
; MN1 Stop On
13149 LD      M2113  ; MN1 Stop On
      ADPRW   H8 H5 H42C H0 H1
      MOV     K0 D616  ; STEP MN1 Move
      AND     M8029  ; Instruction execution complete
      RST     M2113  ; MN1 Stop On
13170 LDF     M2113  ; MN1 Stop On
      SET     M2114  ; MN1 Stop Off
; MN1 Stop Off
13175 LD      M2114  ; MN1 Stop Off
      ADPRW   H8 H5 H42C H0 H0
      AND     M8029  ; Instruction execution complete
      RST     M2114  ; MN1 Stop Off
13191 LDP     M6545  ; PB HMI MN1 Alarm Reset On
      ORP     M1299  ; ALL-ARST
      ORP     M3530  ; TRIG ALARM RESET MN1
      SET     M2115  ; MN1 Alarm Reset On
; MN1 Alarm Reset On
13201 LD      M2115  ; MN1 Alarm Reset On
      ADPRW   H8 H5 H407 H0 H1
      AND     M8029  ; Instruction execution complete
      RST     M2115  ; MN1 Alarm Reset On
13217 LDF     M2115  ; MN1 Alarm Reset On
      SET     M2116  ; MN1 Alarm Reset Off
; MN1 Alarm Reset Off
13222 LD      M2116  ; MN1 Alarm Reset Off
      ADPRW   H8 H5 H407 H0 H0
      AND     M8029  ; Instruction execution complete
      RST     M2116  ; MN1 Alarm Reset Off
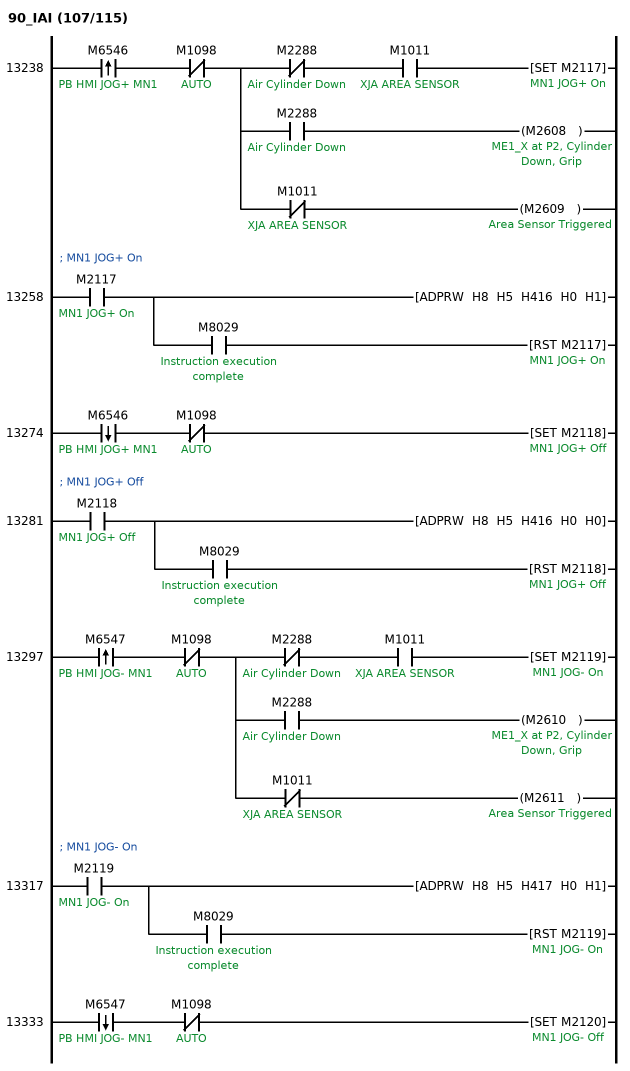
13238 LDP     M6546  ; PB HMI JOG+ MN1
      ANI     M1098  ; AUTO
      MPS
      ANI     M2288  ; Air Cylinder Down
      AND     M1011  ; XJA AREA SENSOR
      SET     M2117  ; MN1 JOG+ On
      MRD
      AND     M2288  ; Air Cylinder Down
      OUT     M2608  ; ME1_X at P2, Cylinder Down, Grip
      MPP
      ANI     M1011  ; XJA AREA SENSOR
      OUT     M2609  ; Area Sensor Triggered
; MN1 JOG+ On
13258 LD      M2117  ; MN1 JOG+ On
      ADPRW   H8 H5 H416 H0 H1
      AND     M8029  ; Instruction execution complete
      RST     M2117  ; MN1 JOG+ On
13274 LDF     M6546  ; PB HMI JOG+ MN1
      ANI     M1098  ; AUTO
      SET     M2118  ; MN1 JOG+ Off
; MN1 JOG+ Off
13281 LD      M2118  ; MN1 JOG+ Off
      ADPRW   H8 H5 H416 H0 H0
      AND     M8029  ; Instruction execution complete
      RST     M2118  ; MN1 JOG+ Off
13297 LDP     M6547  ; PB HMI JOG- MN1
      ANI     M1098  ; AUTO
      MPS
      ANI     M2288  ; Air Cylinder Down
      AND     M1011  ; XJA AREA SENSOR
      SET     M2119  ; MN1 JOG- On
      MRD
      AND     M2288  ; Air Cylinder Down
      OUT     M2610  ; ME1_X at P2, Cylinder Down, Grip
      MPP
      ANI     M1011  ; XJA AREA SENSOR
      OUT     M2611  ; Area Sensor Triggered
; MN1 JOG- On
13317 LD      M2119  ; MN1 JOG- On
      ADPRW   H8 H5 H417 H0 H1
      AND     M8029  ; Instruction execution complete
      RST     M2119  ; MN1 JOG- On
13333 LDF     M6547  ; PB HMI JOG- MN1
      ANI     M1098  ; AUTO
      SET     M2120  ; MN1 JOG- Off
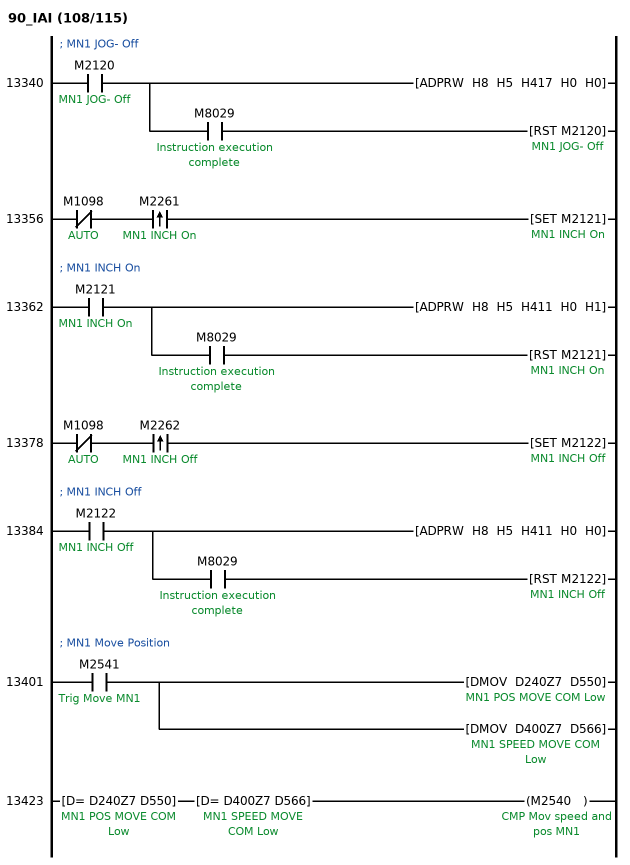
; MN1 JOG- Off
13340 LD      M2120  ; MN1 JOG- Off
      ADPRW   H8 H5 H417 H0 H0
      AND     M8029  ; Instruction execution complete
      RST     M2120  ; MN1 JOG- Off
13356 LDI     M1098  ; AUTO
      ANDP    M2261  ; MN1 INCH On
      SET     M2121  ; MN1 INCH On
; MN1 INCH On
13362 LD      M2121  ; MN1 INCH On
      ADPRW   H8 H5 H411 H0 H1
      AND     M8029  ; Instruction execution complete
      RST     M2121  ; MN1 INCH On
13378 LDI     M1098  ; AUTO
      ANDP    M2262  ; MN1 INCH Off
      SET     M2122  ; MN1 INCH Off
; MN1 INCH Off
13384 LD      M2122  ; MN1 INCH Off
      ADPRW   H8 H5 H411 H0 H0
      AND     M8029  ; Instruction execution complete
      RST     M2122  ; MN1 INCH Off
; MN1 Move Position
13401 LD      M2541  ; Trig Move MN1
      DMOV    D240Z7 D550
        [note] Position
      DMOV    D400Z7 D566
        [note] Speed
13423 LDD=    D240Z7 D550  ; MN1 POS MOVE COM Low
      ANDD=   D400Z7 D566  ; MN1 SPEED MOVE COM Low
      OUT     M2540  ; CMP Mov speed and pos MN1
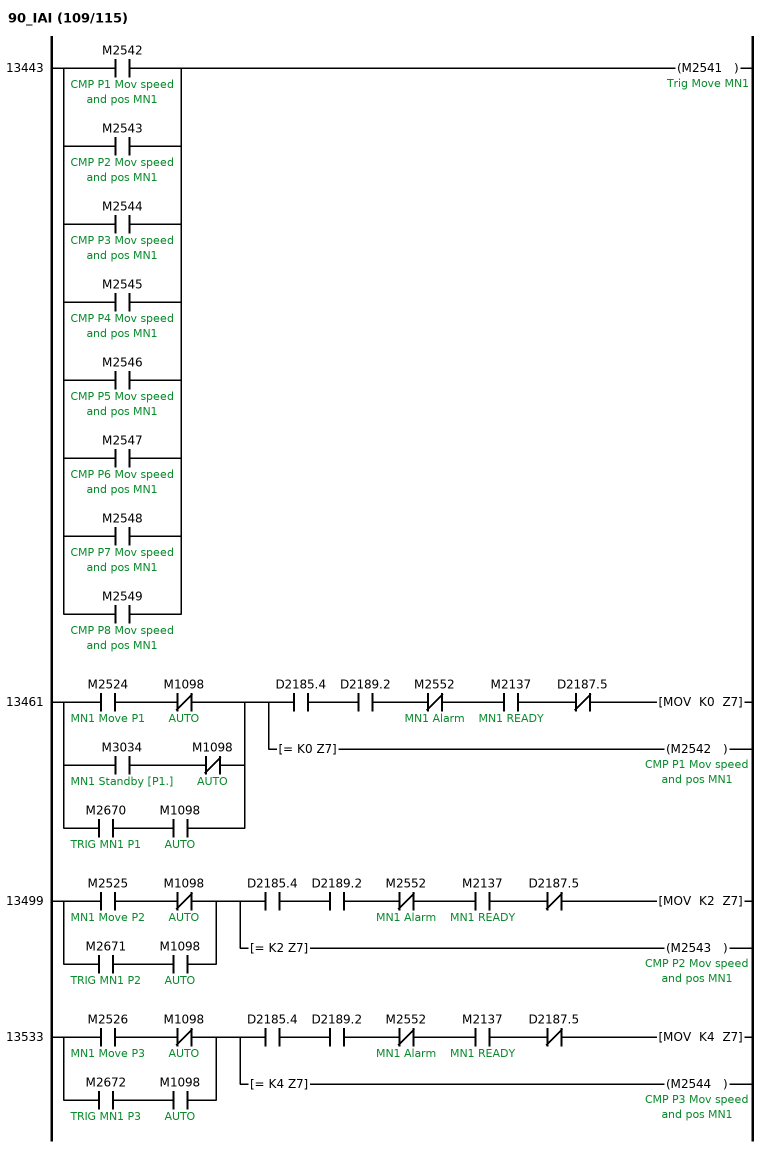
13443 LD      M2542  ; CMP P1 Mov speed and pos MN1
      OR      M2543  ; CMP P2 Mov speed and pos MN1
      OR      M2544  ; CMP P3 Mov speed and pos MN1
      OR      M2545  ; CMP P4 Mov speed and pos MN1
      OR      M2546  ; CMP P5 Mov speed and pos MN1
      OR      M2547  ; CMP P6 Mov speed and pos MN1
      OR      M2548  ; CMP P7 Mov speed and pos MN1
      OR      M2549  ; CMP P8 Mov speed and pos MN1
      OUT     M2541  ; Trig Move MN1
13461 LD      M2524  ; MN1 Move P1
      ANI     M1098  ; AUTO
      LD      M3034  ; MN1 Standby [P1.]
      ANI     M1098  ; AUTO
      ORB
      LD      M2670  ; TRIG MN1 P1
      AND     M1098  ; AUTO
      ORB
      MPS
      AND     D2185.4
      AND     D2189.2
      ANI     M2552  ; MN1 Alarm
      AND     M2137  ; MN1 READY
      ANI     D2187.5
      MOV     K0 Z7
      MPP
      AND=    K0 Z7
      OUT     M2542  ; CMP P1 Mov speed and pos MN1
13499 LD      M2525  ; MN1 Move P2
      ANI     M1098  ; AUTO
      LD      M2671  ; TRIG MN1 P2
      AND     M1098  ; AUTO
      ORB
      MPS
      AND     D2185.4
      AND     D2189.2
      ANI     M2552  ; MN1 Alarm
      AND     M2137  ; MN1 READY
      ANI     D2187.5
      MOV     K2 Z7
      MPP
      AND=    K2 Z7
      OUT     M2543  ; CMP P2 Mov speed and pos MN1
13533 LD      M2526  ; MN1 Move P3
      ANI     M1098  ; AUTO
      LD      M2672  ; TRIG MN1 P3
      AND     M1098  ; AUTO
      ORB
      MPS
      AND     D2185.4
      AND     D2189.2
      ANI     M2552  ; MN1 Alarm
      AND     M2137  ; MN1 READY
      ANI     D2187.5
      MOV     K4 Z7
      MPP
      AND=    K4 Z7
      OUT     M2544  ; CMP P3 Mov speed and pos MN1
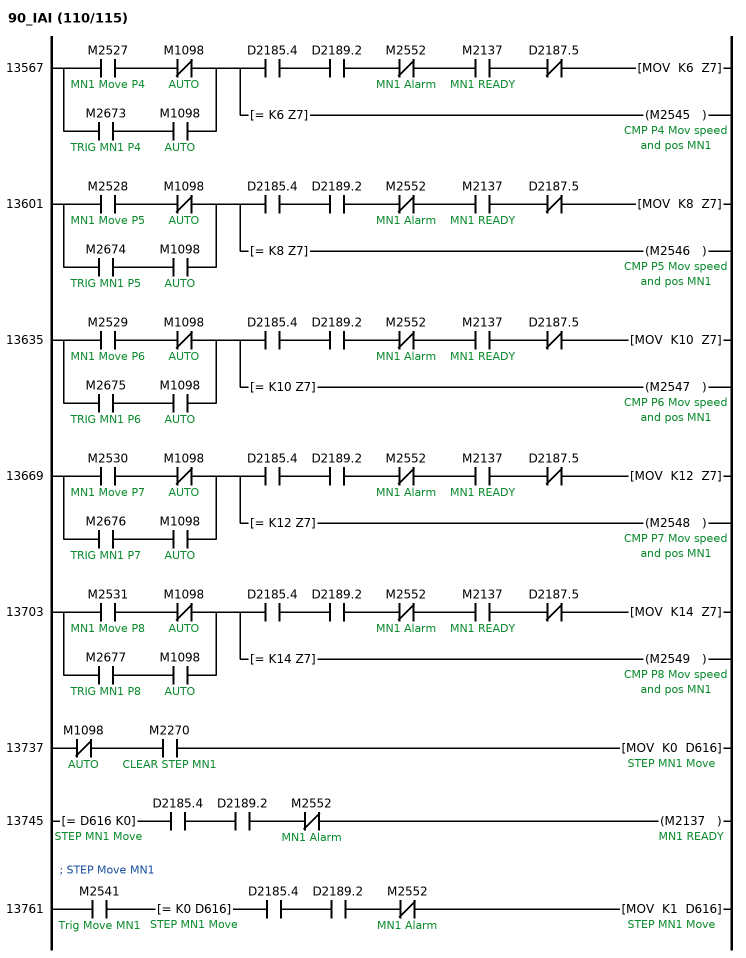
13567 LD      M2527  ; MN1 Move P4
      ANI     M1098  ; AUTO
      LD      M2673  ; TRIG MN1 P4
      AND     M1098  ; AUTO
      ORB
      MPS
      AND     D2185.4
      AND     D2189.2
      ANI     M2552  ; MN1 Alarm
      AND     M2137  ; MN1 READY
      ANI     D2187.5
      MOV     K6 Z7
      MPP
      AND=    K6 Z7
      OUT     M2545  ; CMP P4 Mov speed and pos MN1
13601 LD      M2528  ; MN1 Move P5
      ANI     M1098  ; AUTO
      LD      M2674  ; TRIG MN1 P5
      AND     M1098  ; AUTO
      ORB
      MPS
      AND     D2185.4
      AND     D2189.2
      ANI     M2552  ; MN1 Alarm
      AND     M2137  ; MN1 READY
      ANI     D2187.5
      MOV     K8 Z7
      MPP
      AND=    K8 Z7
      OUT     M2546  ; CMP P5 Mov speed and pos MN1
13635 LD      M2529  ; MN1 Move P6
      ANI     M1098  ; AUTO
      LD      M2675  ; TRIG MN1 P6
      AND     M1098  ; AUTO
      ORB
      MPS
      AND     D2185.4
      AND     D2189.2
      ANI     M2552  ; MN1 Alarm
      AND     M2137  ; MN1 READY
      ANI     D2187.5
      MOV     K10 Z7
      MPP
      AND=    K10 Z7
      OUT     M2547  ; CMP P6 Mov speed and pos MN1
13669 LD      M2530  ; MN1 Move P7
      ANI     M1098  ; AUTO
      LD      M2676  ; TRIG MN1 P7
      AND     M1098  ; AUTO
      ORB
      MPS
      AND     D2185.4
      AND     D2189.2
      ANI     M2552  ; MN1 Alarm
      AND     M2137  ; MN1 READY
      ANI     D2187.5
      MOV     K12 Z7
      MPP
      AND=    K12 Z7
      OUT     M2548  ; CMP P7 Mov speed and pos MN1
13703 LD      M2531  ; MN1 Move P8
      ANI     M1098  ; AUTO
      LD      M2677  ; TRIG MN1 P8
      AND     M1098  ; AUTO
      ORB
      MPS
      AND     D2185.4
      AND     D2189.2
      ANI     M2552  ; MN1 Alarm
      AND     M2137  ; MN1 READY
      ANI     D2187.5
      MOV     K14 Z7
      MPP
      AND=    K14 Z7
      OUT     M2549  ; CMP P8 Mov speed and pos MN1
13737 LDI     M1098  ; AUTO
      AND     M2270  ; CLEAR STEP MN1
      MOV     K0 D616
13745 LD=     D616 K0  ; STEP MN1 Move
      AND     D2185.4
      AND     D2189.2
      ANI     M2552  ; MN1 Alarm
      OUT     M2137  ; MN1 READY
; STEP Move MN1
13761 LD      M2541  ; Trig Move MN1
      AND=    K0 D616  ; STEP MN1 Move
      AND     D2185.4
      AND     D2189.2
      ANI     M2552  ; MN1 Alarm
      MOV     K1 D616
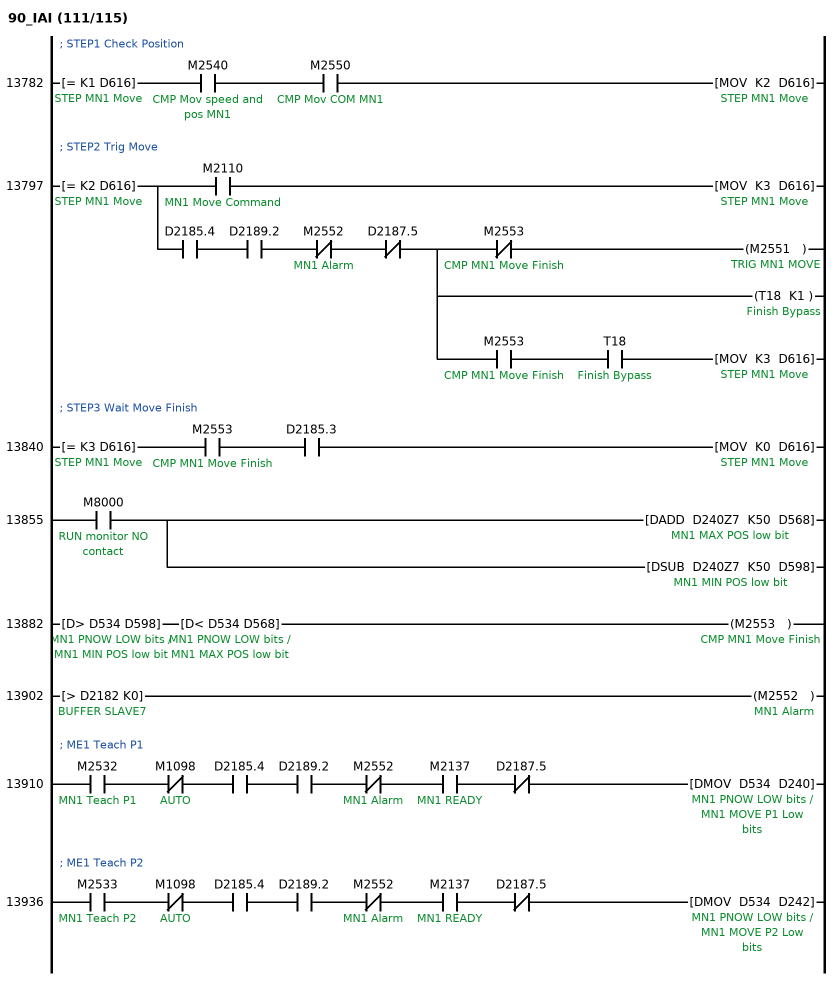
; STEP1 Check Position
13782 LD=     K1 D616  ; STEP MN1 Move
      AND     M2540  ; CMP Mov speed and pos MN1
      AND     M2550  ; CMP Mov COM MN1
      MOV     K2 D616
; STEP2 Trig Move
13797 LD=     K2 D616  ; STEP MN1 Move
      MPS
      AND     M2110  ; MN1 Move Command
      MOV     K3 D616
      MPP
      AND     D2185.4
      AND     D2189.2
      ANI     M2552  ; MN1 Alarm
      ANI     D2187.5
      MPS
      ANI     M2553  ; CMP MN1 Move Finish
      OUT     M2551  ; TRIG MN1 MOVE
      MPP
      OUT     T18 K1  ; Finish Bypass
      AND     M2553  ; CMP MN1 Move Finish
      AND     T18  ; Finish Bypass
      MOV     K3 D616
; STEP3 Wait Move Finish
13840 LD=     K3 D616  ; STEP MN1 Move
      AND     M2553  ; CMP MN1 Move Finish
      AND     D2185.3
      MOV     K0 D616
13855 LD      M8000  ; RUN monitor NO contact
      DADD    D240Z7 K50 D568  ; MN1 MAX POS low bit
      DSUB    D240Z7 K50 D598  ; MN1 MIN POS low bit
13882 LDD>    D534 D598  ; MN1 PNOW LOW bits / MN1 MIN POS low bit
      ANDD<   D534 D568  ; MN1 PNOW LOW bits / MN1 MAX POS low bit
      OUT     M2553  ; CMP MN1 Move Finish
13902 LD>     D2182 K0  ; BUFFER SLAVE7
      OUT     M2552  ; MN1 Alarm
; ME1 Teach P1
13910 LD      M2532  ; MN1 Teach P1
      ANI     M1098  ; AUTO
      AND     D2185.4
      AND     D2189.2
      ANI     M2552  ; MN1 Alarm
      AND     M2137  ; MN1 READY
      ANI     D2187.5
      DMOV    D534 D240  ; MN1 MOVE P1 Low bits
; ME1 Teach P2
13936 LD      M2533  ; MN1 Teach P2
      ANI     M1098  ; AUTO
      AND     D2185.4
      AND     D2189.2
      ANI     M2552  ; MN1 Alarm
      AND     M2137  ; MN1 READY
      ANI     D2187.5
      DMOV    D534 D242  ; MN1 MOVE P2 Low bits
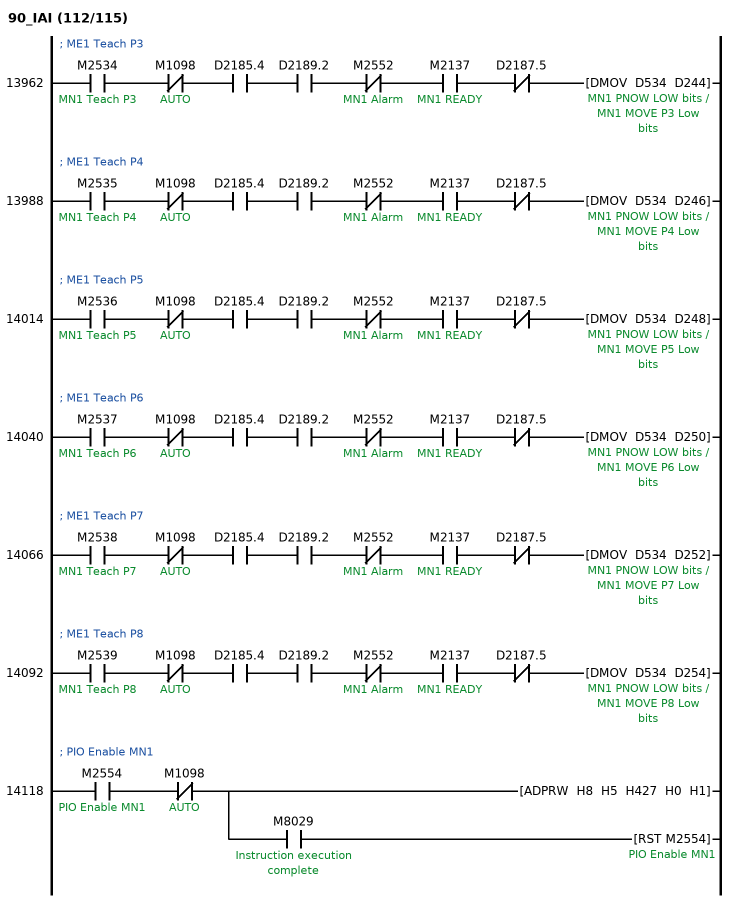
; ME1 Teach P3
13962 LD      M2534  ; MN1 Teach P3
      ANI     M1098  ; AUTO
      AND     D2185.4
      AND     D2189.2
      ANI     M2552  ; MN1 Alarm
      AND     M2137  ; MN1 READY
      ANI     D2187.5
      DMOV    D534 D244  ; MN1 MOVE P3 Low bits
; ME1 Teach P4
13988 LD      M2535  ; MN1 Teach P4
      ANI     M1098  ; AUTO
      AND     D2185.4
      AND     D2189.2
      ANI     M2552  ; MN1 Alarm
      AND     M2137  ; MN1 READY
      ANI     D2187.5
      DMOV    D534 D246  ; MN1 MOVE P4 Low bits
; ME1 Teach P5
14014 LD      M2536  ; MN1 Teach P5
      ANI     M1098  ; AUTO
      AND     D2185.4
      AND     D2189.2
      ANI     M2552  ; MN1 Alarm
      AND     M2137  ; MN1 READY
      ANI     D2187.5
      DMOV    D534 D248  ; MN1 MOVE P5 Low bits
; ME1 Teach P6
14040 LD      M2537  ; MN1 Teach P6
      ANI     M1098  ; AUTO
      AND     D2185.4
      AND     D2189.2
      ANI     M2552  ; MN1 Alarm
      AND     M2137  ; MN1 READY
      ANI     D2187.5
      DMOV    D534 D250  ; MN1 MOVE P6 Low bits
; ME1 Teach P7
14066 LD      M2538  ; MN1 Teach P7
      ANI     M1098  ; AUTO
      AND     D2185.4
      AND     D2189.2
      ANI     M2552  ; MN1 Alarm
      AND     M2137  ; MN1 READY
      ANI     D2187.5
      DMOV    D534 D252  ; MN1 MOVE P7 Low bits
; ME1 Teach P8
14092 LD      M2539  ; MN1 Teach P8
      ANI     M1098  ; AUTO
      AND     D2185.4
      AND     D2189.2
      ANI     M2552  ; MN1 Alarm
      AND     M2137  ; MN1 READY
      ANI     D2187.5
      DMOV    D534 D254  ; MN1 MOVE P8 Low bits
; PIO Enable MN1
14118 LD      M2554  ; PIO Enable MN1
      ANI     M1098  ; AUTO
      ADPRW   H8 H5 H427 H0 H1
      AND     M8029  ; Instruction execution complete
      RST     M2554  ; PIO Enable MN1
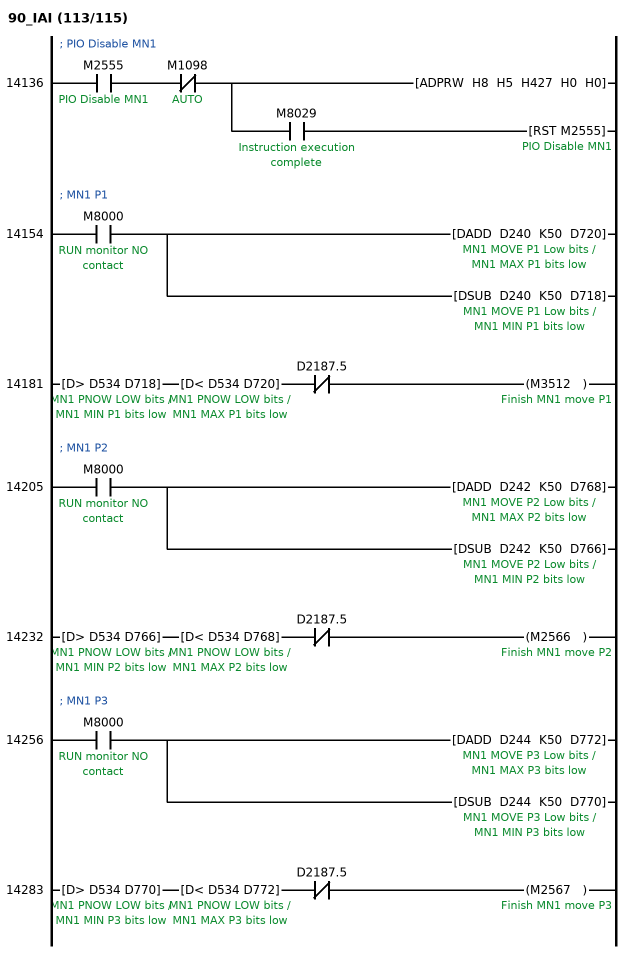
; PIO Disable MN1
14136 LD      M2555  ; PIO Disable MN1
      ANI     M1098  ; AUTO
      ADPRW   H8 H5 H427 H0 H0
      AND     M8029  ; Instruction execution complete
      RST     M2555  ; PIO Disable MN1
; MN1 P1
14154 LD      M8000  ; RUN monitor NO contact
      DADD    D240 K50 D720  ; MN1 MAX P1 bits low
      DSUB    D240 K50 D718  ; MN1 MIN P1 bits low
14181 LDD>    D534 D718  ; MN1 PNOW LOW bits / MN1 MIN P1 bits low
      ANDD<   D534 D720  ; MN1 PNOW LOW bits / MN1 MAX P1 bits low
      ANI     D2187.5
      OUT     M3512  ; Finish MN1 move P1
; MN1 P2
14205 LD      M8000  ; RUN monitor NO contact
      DADD    D242 K50 D768  ; MN1 MAX P2 bits low
      DSUB    D242 K50 D766  ; MN1 MIN P2 bits low
14232 LDD>    D534 D766  ; MN1 PNOW LOW bits / MN1 MIN P2 bits low
      ANDD<   D534 D768  ; MN1 PNOW LOW bits / MN1 MAX P2 bits low
      ANI     D2187.5
      OUT     M2566  ; Finish MN1 move P2
; MN1 P3
14256 LD      M8000  ; RUN monitor NO contact
      DADD    D244 K50 D772  ; MN1 MAX P3 bits low
      DSUB    D244 K50 D770  ; MN1 MIN P3 bits low
14283 LDD>    D534 D770  ; MN1 PNOW LOW bits / MN1 MIN P3 bits low
      ANDD<   D534 D772  ; MN1 PNOW LOW bits / MN1 MAX P3 bits low
      ANI     D2187.5
      OUT     M2567  ; Finish MN1 move P3
